// TIA Portal V17 export
// export: Created 2023-02-26T22:57:58.8768627Z, ExportSetting WithDefaults, DisplayName Totally Integrated Automation Portal, DisplayVersion V17, DisplayName TIA Portal Openness, DisplayVersion V17, DisplayName TIA Portal Version Control Interface, DisplayVersion V17, DisplayName TIA Portal Test Suite Advanced, DisplayVersion V17, DisplayName STEP 7 Professional, DisplayVersion V17, DisplayName SIMATIC Energy Suite, DisplayVersion V17, DisplayName STEP 7 Safety, DisplayVersion V17, DisplayName WinCC Professional, DisplayVersion V17
FUNCTION_BLOCK "LOG_CountMode"   // FB3, LAD
{ S7_Optimized_Access := 'TRUE' }
VERSION : 0.1
// stored: AutoNumber true, IsIECCheckEnabled false, IsRetainMemResEnabled false, MemoryReserve 100, SetENOAutomatically false, UDAEnableTagReadback false
   VAR_INPUT
      "StartLine/StopLine" : Bool;
      Mode : Bool;
   END_VAR
   VAR_IN_OUT
      QMode : UDInt;
   END_VAR
   VAR
      P_Mode : Bool;
   END_VAR
   VAR_TEMP   // added for the SCL form of the ladder/FBD networks
      _w1 : Bool;
   END_VAR
BEGIN

REGION Network 1
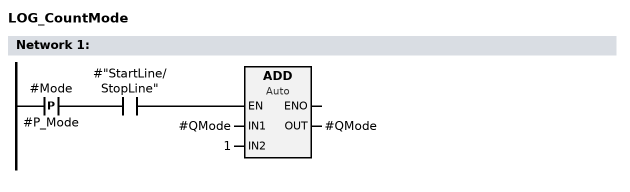
   RUNG wire#powerrail
      P_Contact(operand := #Mode, bit := #P_Mode)
      Contact( #"StartLine/StopLine" )
      { S7_GenerateENO := "TRUE" } Add(in1 := #QMode, in2 := 1, out => #QMode)
   END_RUNG
   // the same network as SCL:
   #_w1 := #Mode AND NOT #P_Mode;   // rising edge of #Mode
   #P_Mode := #Mode;
   IF #_w1 AND #"StartLine/StopLine" THEN #QMode := #QMode + 1; END_IF;
END_REGION
END_FUNCTION_BLOCK
